// TwinCAT 3 PLC project pyads_sample
// ProgramVersion: 3.1.4024.0
// libraries:
//   Tc2_Standard, * (Beckhoff Automation GmbH)
//   Tc2_System, * (Beckhoff Automation GmbH)
//   Tc3_Module, * (Beckhoff Automation GmbH)
// project tree:
//   DUTs/ ST_sample.TcDUT
//   / PlcTask.TcTTO
//   POUs/ MAIN.TcPOU
// real-time tasks:
//   TASK PlcTask: cycle T#250us, priority 20, ADS port 350

CONFIGURATION pyads_sample
    RESOURCE PLC ON TwinCAT3
        TASK PlcTask(INTERVAL := T#250us, PRIORITY := 20);
        PROGRAM MAIN WITH PlcTask : MAIN;
    END_RESOURCE
END_CONFIGURATION

// ---- DUTs/ST_sample.TcDUT
{attribute 'pack_mode' := '1'}
TYPE ST_sample :
STRUCT
	title :STRING;
	name: STRING;
	age: UINT;
	sex: UINT;
	mail_address : STRING;
	event_date : ULINT;
	description : STRING;
END_STRUCT
END_TYPE

// ---- POUs/MAIN.TcPOU
PROGRAM MAIN
VAR

	events : ARRAY [1..5] OF ST_sample := [
		(title := 'Promotion ceremony', name := 'Kenichi Takahashi', age := 10, sex := 1, mail_address := 'ken@example.com', description := 'Pass to the next grade'),
		(title := 'Promotion ceremony', name := 'Takashi Shimizu', age := 18, sex := 1, mail_address := 'takashi@example.com', description := 'Pass to the next grade'),
		(title := 'Promotion ceremony', name := 'Junich Yamada', age := 13, sex := 1, mail_address := 'jun@example.com', description := 'Pass to the next grade'),
		(title := 'Promotion ceremony', name := 'Koichiro Honda', age := 12, sex := 1, mail_address := 'koichi@example.com', description := 'Pass to the next grade'),
		(title := 'Promotion ceremony', name := 'Sojiro Yokota', age := 11, sex := 1, mail_address := 'Sojiro@example.com', description := 'Pass to the next grade')
	];
	
	ads_watch_variable : ST_sample;
	last_dt : ULINT;
	diff_dt : ULINT;
	event_timer :TON;
	i :UINT;
	id : UINT;
END_VAR

event_timer(IN := NOT event_timer.Q, PT := T#10S);

id := id + 1;

IF id = 16#FFFF THEN
	id := 0;
END_IF

//IF event_timer.Q THEN
	IF i < 1 OR i > 5 THEN
		i := 1;
	END_IF
	events[i].age := i + 5;
	ads_watch_variable := events[i];
	ads_watch_variable.event_date := F_GetSystemTime();
	diff_dt := ads_watch_variable.event_date - last_dt;
	last_dt := ads_watch_variable.event_date;
	
	i :=  i + 1;
//END_IF

END_PROGRAM
